INTERFACE I_EventEmitter EXTENDS __SYSTEM.IQueryInterface

METHOD PUBLIC OffEvent
VAR_INPUT
	EventName : T_MaxString;
	EventHandler : I_EventHandler;
END_VAR
END_METHOD

METHOD PUBLIC OnceEvent
VAR_INPUT
	EventName : T_MaxString;
	EventHandler : I_EventHandler;
END_VAR
END_METHOD

METHOD PUBLIC OnEvent
VAR_INPUT
	EventName : T_MaxString;
	EventHandler : I_EventHandler;
END_VAR
END_METHOD

END_INTERFACE

(* stored: Version 1.1.0.1, ProductVersion 3.1.4024.12
   Itf I_EventEmitter: Id {521513c8-a1e5-0eda-336a-353a9fc8fd4a}
   Method OffEvent: Id {5b41fd39-59cc-01d6-1483-4885f4971279}
   Method OnceEvent: Id {6ddfc555-780a-49bd-a30f-34a0808f6006}
   Method OnEvent: Id {b949e301-16ff-080e-090e-4a7708470395} *)
